INTERFACE I_JsonDeserializerDisposedEvent EXTENDS I_Event

PROPERTY PUBLIC Target : I_JsonDeserializer
GET
END_GET
END_PROPERTY

END_INTERFACE

(* stored: Version 1.1.0.1, ProductVersion 3.1.4024.12
   Itf I_JsonDeserializerDisposedEvent: Id {a972cec1-feba-428b-bd7d-6fdf767f8322}
   Property Target: Id {2a98b9fc-5cd3-40b2-84bc-77eaeffa75b7}
   Get Get: Id {4b2b3482-3dd2-422d-ad58-8f38bef2cf82} *)
